// Mitsubishi GX Works2 project: 20160811現状設定   PLC: Q03UDV

PROGRAM P1
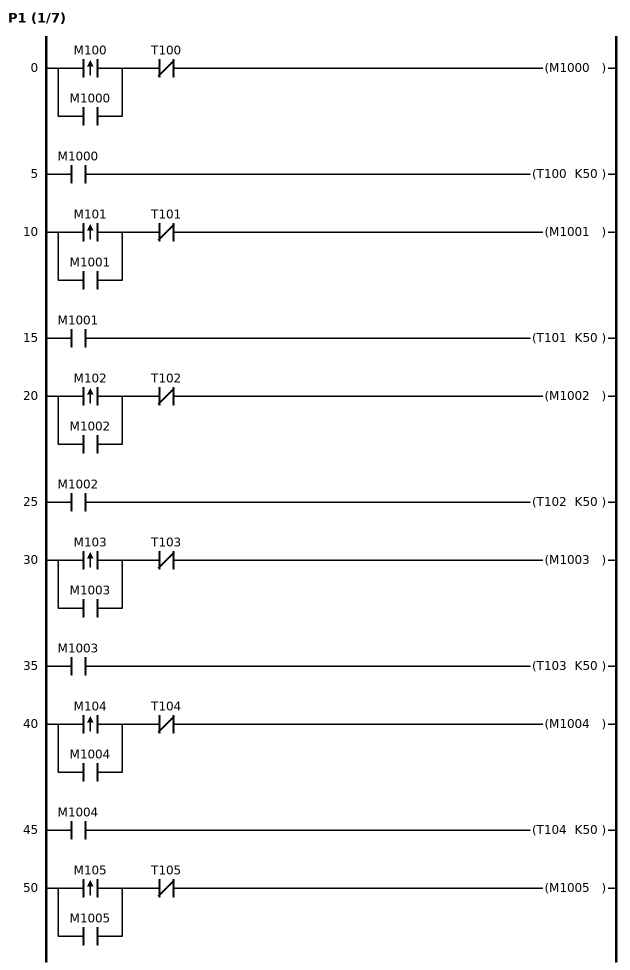
0     LDP     M100
      OR      M1000
      ANI     T100
      OUT     M1000
5     LD      M1000
      OUT     T100 K50
10    LDP     M101
      OR      M1001
      ANI     T101
      OUT     M1001
15    LD      M1001
      OUT     T101 K50
20    LDP     M102
      OR      M1002
      ANI     T102
      OUT     M1002
25    LD      M1002
      OUT     T102 K50
30    LDP     M103
      OR      M1003
      ANI     T103
      OUT     M1003
35    LD      M1003
      OUT     T103 K50
40    LDP     M104
      OR      M1004
      ANI     T104
      OUT     M1004
45    LD      M1004
      OUT     T104 K50
50    LDP     M105
      OR      M1005
      ANI     T105
      OUT     M1005
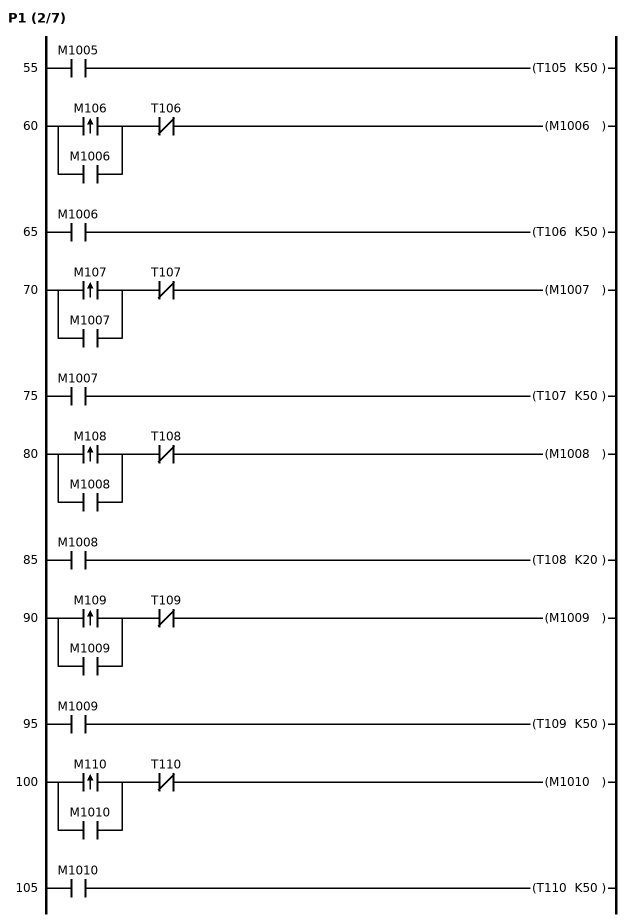
55    LD      M1005
      OUT     T105 K50
60    LDP     M106
      OR      M1006
      ANI     T106
      OUT     M1006
65    LD      M1006
      OUT     T106 K50
70    LDP     M107
      OR      M1007
      ANI     T107
      OUT     M1007
75    LD      M1007
      OUT     T107 K50
80    LDP     M108
      OR      M1008
      ANI     T108
      OUT     M1008
85    LD      M1008
      OUT     T108 K20
90    LDP     M109
      OR      M1009
      ANI     T109
      OUT     M1009
95    LD      M1009
      OUT     T109 K50
100   LDP     M110
      OR      M1010
      ANI     T110
      OUT     M1010
105   LD      M1010
      OUT     T110 K50
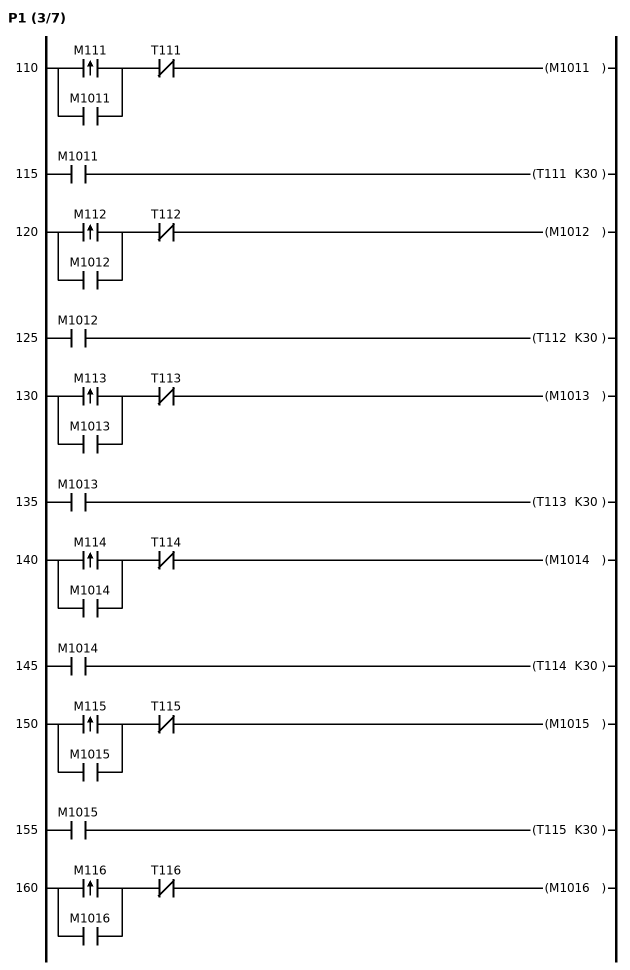
110   LDP     M111
      OR      M1011
      ANI     T111
      OUT     M1011
115   LD      M1011
      OUT     T111 K30
120   LDP     M112
      OR      M1012
      ANI     T112
      OUT     M1012
125   LD      M1012
      OUT     T112 K30
130   LDP     M113
      OR      M1013
      ANI     T113
      OUT     M1013
135   LD      M1013
      OUT     T113 K30
140   LDP     M114
      OR      M1014
      ANI     T114
      OUT     M1014
145   LD      M1014
      OUT     T114 K30
150   LDP     M115
      OR      M1015
      ANI     T115
      OUT     M1015
155   LD      M1015
      OUT     T115 K30
160   LDP     M116
      OR      M1016
      ANI     T116
      OUT     M1016
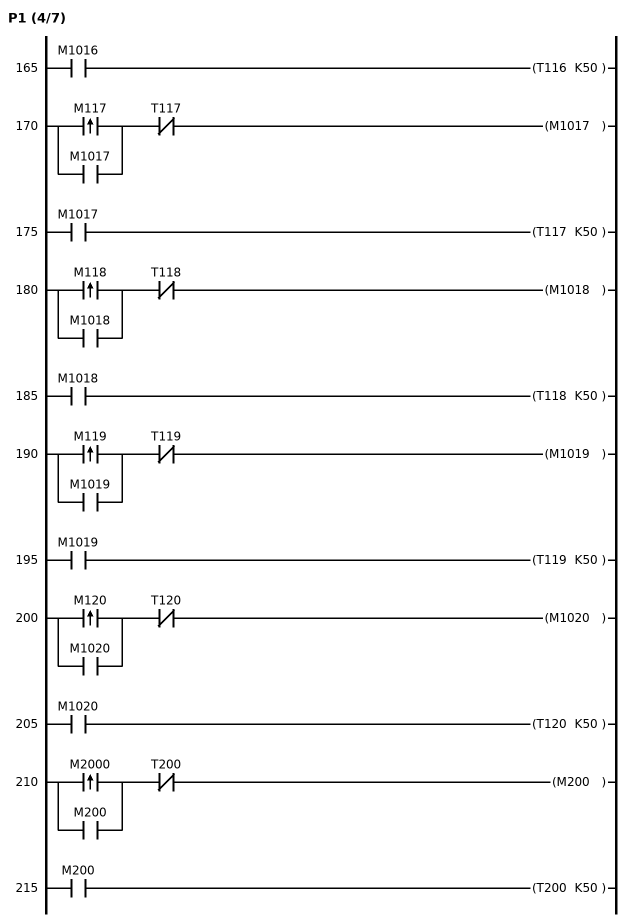
165   LD      M1016
      OUT     T116 K50
170   LDP     M117
      OR      M1017
      ANI     T117
      OUT     M1017
175   LD      M1017
      OUT     T117 K50
180   LDP     M118
      OR      M1018
      ANI     T118
      OUT     M1018
185   LD      M1018
      OUT     T118 K50
190   LDP     M119
      OR      M1019
      ANI     T119
      OUT     M1019
195   LD      M1019
      OUT     T119 K50
200   LDP     M120
      OR      M1020
      ANI     T120
      OUT     M1020
205   LD      M1020
      OUT     T120 K50
210   LDP     M2000
      OR      M200
      ANI     T200
      OUT     M200
215   LD      M200
      OUT     T200 K50
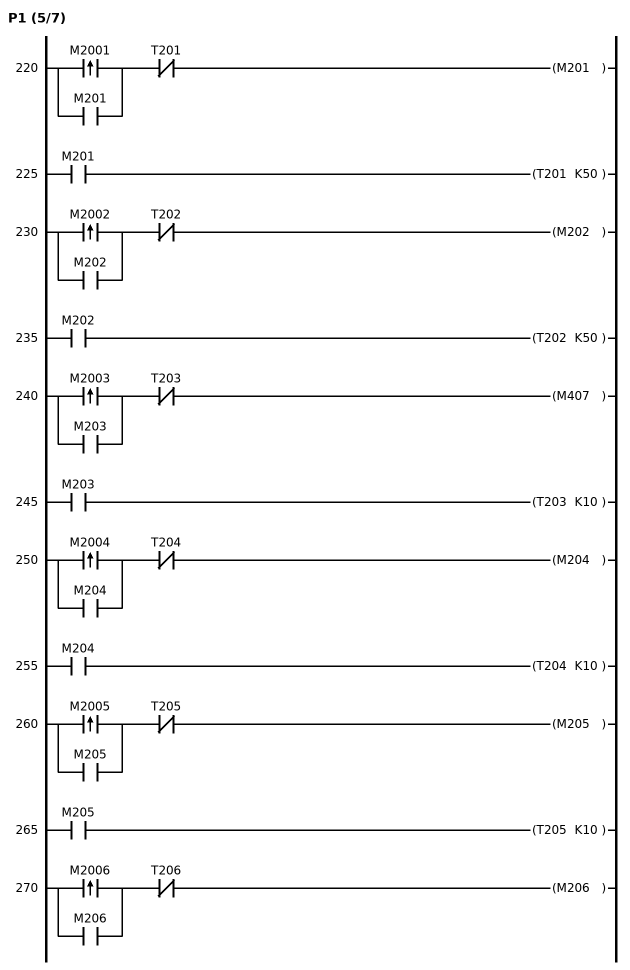
220   LDP     M2001
      OR      M201
      ANI     T201
      OUT     M201
225   LD      M201
      OUT     T201 K50
230   LDP     M2002
      OR      M202
      ANI     T202
      OUT     M202
235   LD      M202
      OUT     T202 K50
240   LDP     M2003
      OR      M203
      ANI     T203
      OUT     M407
245   LD      M203
      OUT     T203 K10
250   LDP     M2004
      OR      M204
      ANI     T204
      OUT     M204
255   LD      M204
      OUT     T204 K10
260   LDP     M2005
      OR      M205
      ANI     T205
      OUT     M205
265   LD      M205
      OUT     T205 K10
270   LDP     M2006
      OR      M206
      ANI     T206
      OUT     M206
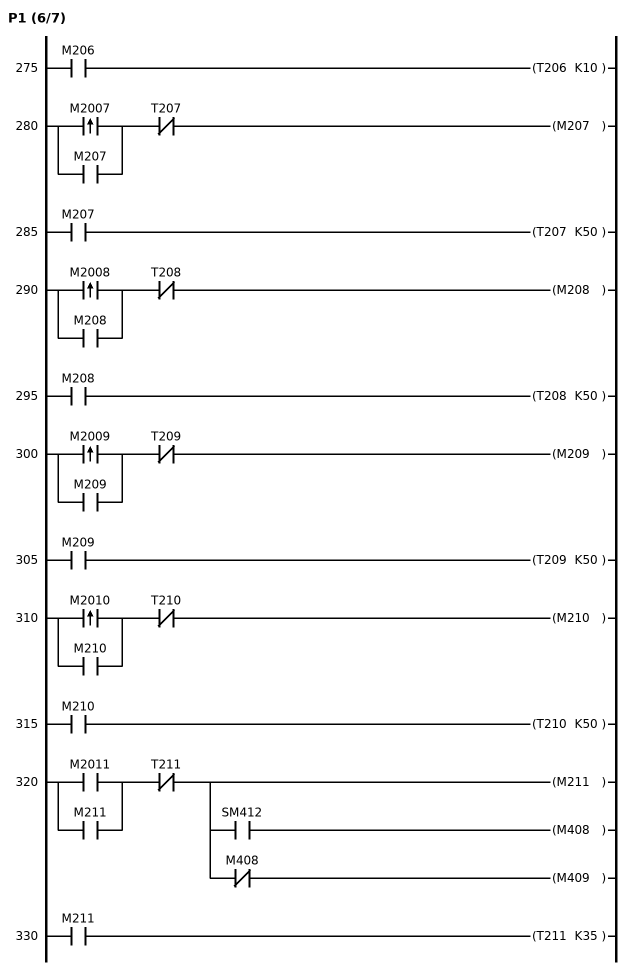
275   LD      M206
      OUT     T206 K10
280   LDP     M2007
      OR      M207
      ANI     T207
      OUT     M207
285   LD      M207
      OUT     T207 K50
290   LDP     M2008
      OR      M208
      ANI     T208
      OUT     M208
295   LD      M208
      OUT     T208 K50
300   LDP     M2009
      OR      M209
      ANI     T209
      OUT     M209
305   LD      M209
      OUT     T209 K50
310   LDP     M2010
      OR      M210
      ANI     T210
      OUT     M210
315   LD      M210
      OUT     T210 K50
320   LD      M2011
      OR      M211
      ANI     T211
      OUT     M211
      MPS
      AND     SM412
      OUT     M408
      MPP
      ANI     M408
      OUT     M409
330   LD      M211
      OUT     T211 K35
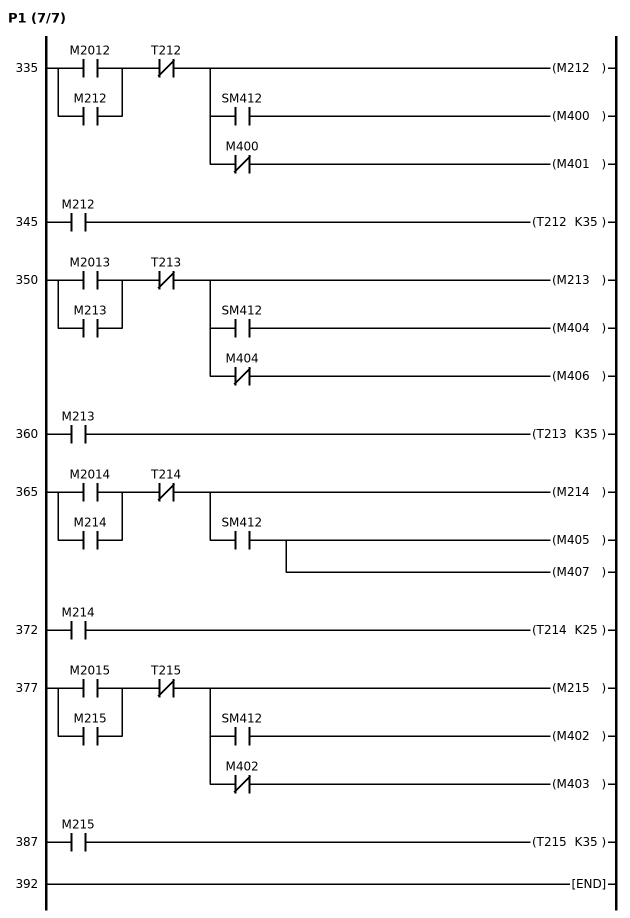
335   LD      M2012
      OR      M212
      ANI     T212
      OUT     M212
      MPS
      AND     SM412
      OUT     M400
      MPP
      ANI     M400
      OUT     M401
345   LD      M212
      OUT     T212 K35
350   LD      M2013
      OR      M213
      ANI     T213
      OUT     M213
      MPS
      AND     SM412
      OUT     M404
      MPP
      ANI     M404
      OUT     M406
360   LD      M213
      OUT     T213 K35
365   LD      M2014
      OR      M214
      ANI     T214
      OUT     M214
      AND     SM412
      OUT     M405
      OUT     M407
372   LD      M214
      OUT     T214 K25
377   LD      M2015
      OR      M215
      ANI     T215
      OUT     M215
      MPS
      AND     SM412
      OUT     M402
      MPP
      ANI     M402
      OUT     M403
387   LD      M215
      OUT     T215 K35
392   END
END_PROGRAM
